// TwinCAT 3 PLC project Standard
// ProgramVersion: 3.1.4023.0
// libraries:
//   Tc2_Standard, * (Beckhoff Automation GmbH)
//   Tc2_System, * (Beckhoff Automation GmbH)
//   Tc3_Module, * (Beckhoff Automation GmbH)
// project tree:
//   / PlcTask.TcTTO
//   POUs/ MAIN.TcPOU
// real-time tasks:
//   TASK PlcTask: cycle T#10ms, priority 20, ADS port 350

CONFIGURATION Standard
    RESOURCE PLC ON TwinCAT3
        TASK PlcTask(INTERVAL := T#10ms, PRIORITY := 20);
        PROGRAM MAIN WITH PlcTask : MAIN;
    END_RESOURCE
END_CONFIGURATION

// ---- POUs/MAIN.TcPOU
PROGRAM MAIN
VAR
	//fbTon : TON := (PT := T#10S);
	//bThisIsABoolean : BOOL;	

	//fbTof : TOF := (PT := T#10S);
	//bThisIsABoolean : BOOL;
	
	//fbRtrig : R_TRIG;
	//bSomeBoolean : BOOL;
	//nTriggerCounter : ULINT;
	
	//fbFtrig : F_TRIG;
	//bSomeBoolean : BOOL;
	//nTriggerCounter : ULINT;
	
	sString1 : STRING(255) := 'Hello';
	sString2 : STRING(255) := 'World';
	sResultString : STRING(255);
END_VAR

//fbTon(in := bThisIsABoolean);
//fbTof(in := bThisIsABoolean);

//fbFtrig(CLK := bSomeBoolean);
//IF fbFtrig.Q THEN
	//nTriggerCounter := nTriggerCounter + 1;
//END_IF

sResultString := CONCAT(STR1 := sString1, STR2 := sString2);

END_PROGRAM
